// TIA Portal V15.1 export
// export: Created 2020-06-12T07:35:52.2724609Z, ExportSetting None, DisplayName Totally Integrated Automation Portal, DisplayVersion V15.1, DisplayName TIA Portal Openness, DisplayVersion V15.1, DisplayName STEP 7 Professional, DisplayVersion V15.1, DisplayName STEP 7 Safety, DisplayVersion V15.1, DisplayName WinCC Advanced, DisplayVersion V15.1
FUNCTION "MELT_Curves" : Void   // FC224, FBD
TITLE = Melt curves management
{ S7_Optimized_Access := 'FALSE' }
// stored: SetENOAutomatically False
   VAR_TEMP
      tMode : Int;
      tPmax : Real;
      tImax : Real;
      tIdx : Int;
      tDoCheck : Bool;
      tHTRelPower : Real;
      i : Int;
      tX : Real;
      tZ : Real;
      tR : Real;
      tPF : Real;
      tRslag : Real;
      tIset : Real;
      tUmin : Real;
      tUmax : Real;
   END_VAR
BEGIN

REGION Network 1: Staring resistance curve
   // Swing controller will be activatied during start phase, after time delay. After 
   // this the Resistance curve will be frosen
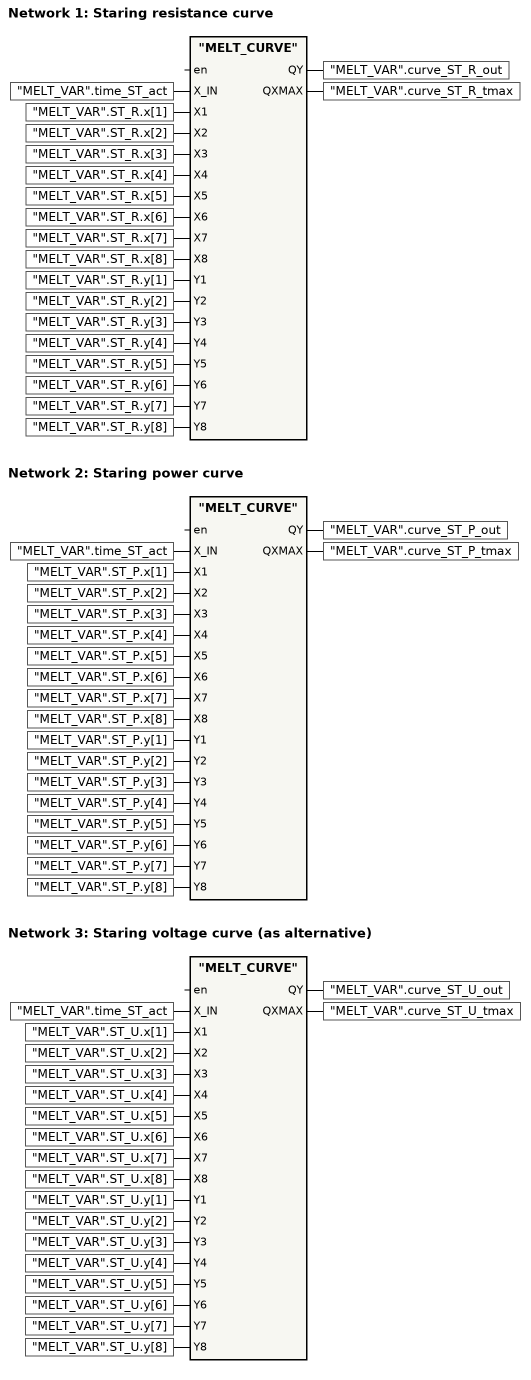
   "MELT_CURVE"(X_IN := "MELT_VAR".time_ST_act,
                X1 := "MELT_VAR".ST_R.x[1],
                X2 := "MELT_VAR".ST_R.x[2],
                X3 := "MELT_VAR".ST_R.x[3],
                X4 := "MELT_VAR".ST_R.x[4],
                X5 := "MELT_VAR".ST_R.x[5],
                X6 := "MELT_VAR".ST_R.x[6],
                X7 := "MELT_VAR".ST_R.x[7],
                X8 := "MELT_VAR".ST_R.x[8],
                Y1 := "MELT_VAR".ST_R.y[1],
                Y2 := "MELT_VAR".ST_R.y[2],
                Y3 := "MELT_VAR".ST_R.y[3],
                Y4 := "MELT_VAR".ST_R.y[4],
                Y5 := "MELT_VAR".ST_R.y[5],
                Y6 := "MELT_VAR".ST_R.y[6],
                Y7 := "MELT_VAR".ST_R.y[7],
                Y8 := "MELT_VAR".ST_R.y[8],
                QY => "MELT_VAR".curve_ST_R_out,
                QXMAX => "MELT_VAR".curve_ST_R_tmax);
END_REGION

REGION Network 2: Staring power curve
   "MELT_CURVE"(X_IN := "MELT_VAR".time_ST_act,
                X1 := "MELT_VAR".ST_P.x[1],
                X2 := "MELT_VAR".ST_P.x[2],
                X3 := "MELT_VAR".ST_P.x[3],
                X4 := "MELT_VAR".ST_P.x[4],
                X5 := "MELT_VAR".ST_P.x[5],
                X6 := "MELT_VAR".ST_P.x[6],
                X7 := "MELT_VAR".ST_P.x[7],
                X8 := "MELT_VAR".ST_P.x[8],
                Y1 := "MELT_VAR".ST_P.y[1],
                Y2 := "MELT_VAR".ST_P.y[2],
                Y3 := "MELT_VAR".ST_P.y[3],
                Y4 := "MELT_VAR".ST_P.y[4],
                Y5 := "MELT_VAR".ST_P.y[5],
                Y6 := "MELT_VAR".ST_P.y[6],
                Y7 := "MELT_VAR".ST_P.y[7],
                Y8 := "MELT_VAR".ST_P.y[8],
                QY => "MELT_VAR".curve_ST_P_out,
                QXMAX => "MELT_VAR".curve_ST_P_tmax);
END_REGION

REGION Network 3: Staring voltage curve (as alternative)
   "MELT_CURVE"(X_IN := "MELT_VAR".time_ST_act,
                X1 := "MELT_VAR".ST_U.x[1],
                X2 := "MELT_VAR".ST_U.x[2],
                X3 := "MELT_VAR".ST_U.x[3],
                X4 := "MELT_VAR".ST_U.x[4],
                X5 := "MELT_VAR".ST_U.x[5],
                X6 := "MELT_VAR".ST_U.x[6],
                X7 := "MELT_VAR".ST_U.x[7],
                X8 := "MELT_VAR".ST_U.x[8],
                Y1 := "MELT_VAR".ST_U.y[1],
                Y2 := "MELT_VAR".ST_U.y[2],
                Y3 := "MELT_VAR".ST_U.y[3],
                Y4 := "MELT_VAR".ST_U.y[4],
                Y5 := "MELT_VAR".ST_U.y[5],
                Y6 := "MELT_VAR".ST_U.y[6],
                Y7 := "MELT_VAR".ST_U.y[7],
                Y8 := "MELT_VAR".ST_U.y[8],
                QY => "MELT_VAR".curve_ST_U_out,
                QXMAX => "MELT_VAR".curve_ST_U_tmax);
END_REGION

REGION Network 4: Internal inducatnce
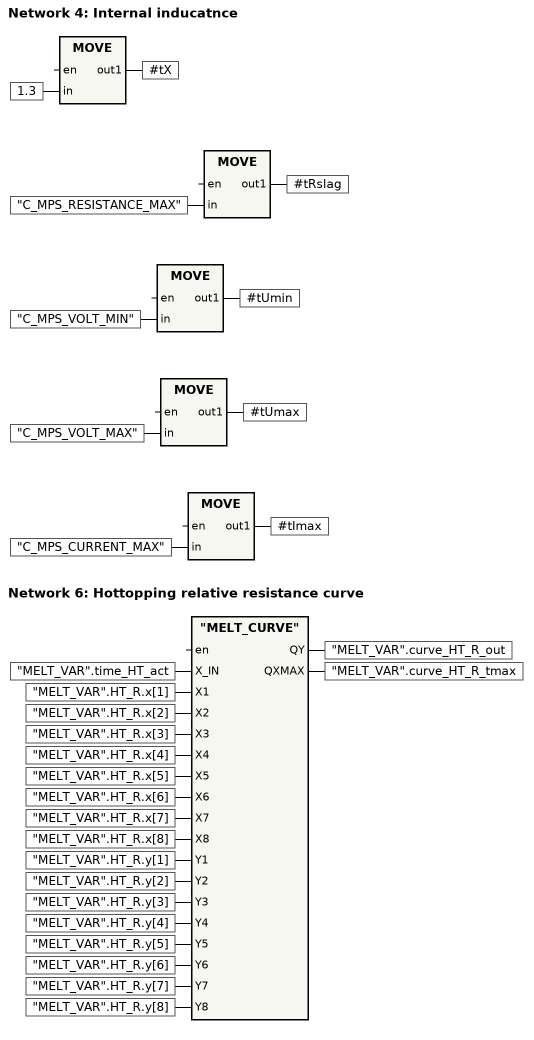
   #tX := 1.3;
   #tRslag := "C_MPS_RESISTANCE_MAX";
   #tUmin := "C_MPS_VOLT_MIN";
   #tUmax := "C_MPS_VOLT_MAX";
   #tImax := "C_MPS_CURRENT_MAX";
END_REGION

REGION Network 5 (SCL): Recaclulate the starting curve: (P,R) -> (U,R)
   IF "MELT_VAR".use_recalc_u THEN
       #tIset := 10.0;
       FOR #i := 1 TO 8 DO
       #tR := "MELT_VAR".ST_R.y[#i];
       #tZ := #tR + #tX;
       #tPF := #tR / #tZ;
       "PUR_CONSTR"(iEnable:=true,
                    iMode:=2,
                    iCosPhi:=#tPF,
                    iRslag:=#tRslag,
                    pQmax:=3500.0,
                    pUmin:=#tUmin,
                    pUmax:=#tUmax,
                    pImax:=#tImax,
                    qPmax=>#tPmax,
                    qImax=>#tImax,
                    ioPset:="MELT_VAR".ST_P.y[#i],
                    ioRset:="MELT_VAR".ST_R.y[#i],
                    ioUset:="MELT_VAR".ST_U.y[#i],
                    ioIset:=#tIset);

       END_FOR;
   END_IF;
END_REGION

REGION Network 6: Hottopping relative resistance curve
   "MELT_CURVE"(X_IN := "MELT_VAR".time_HT_act,
                X1 := "MELT_VAR".HT_R.x[1],
                X2 := "MELT_VAR".HT_R.x[2],
                X3 := "MELT_VAR".HT_R.x[3],
                X4 := "MELT_VAR".HT_R.x[4],
                X5 := "MELT_VAR".HT_R.x[5],
                X6 := "MELT_VAR".HT_R.x[6],
                X7 := "MELT_VAR".HT_R.x[7],
                X8 := "MELT_VAR".HT_R.x[8],
                Y1 := "MELT_VAR".HT_R.y[1],
                Y2 := "MELT_VAR".HT_R.y[2],
                Y3 := "MELT_VAR".HT_R.y[3],
                Y4 := "MELT_VAR".HT_R.y[4],
                Y5 := "MELT_VAR".HT_R.y[5],
                Y6 := "MELT_VAR".HT_R.y[6],
                Y7 := "MELT_VAR".HT_R.y[7],
                Y8 := "MELT_VAR".HT_R.y[8],
                QY => "MELT_VAR".curve_HT_R_out,
                QXMAX => "MELT_VAR".curve_HT_R_tmax);
END_REGION

REGION Network 7: Hottopping relative power curve
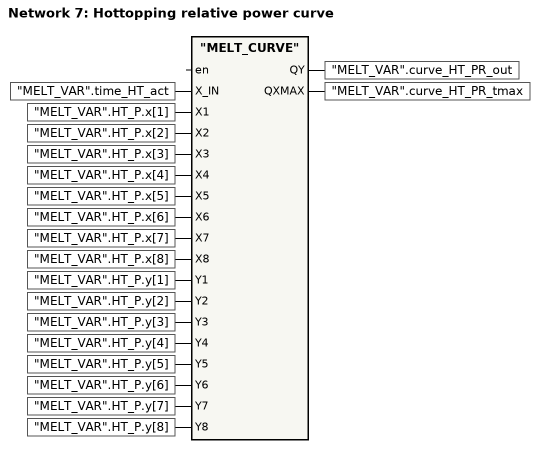
   "MELT_CURVE"(X_IN := "MELT_VAR".time_HT_act,
                X1 := "MELT_VAR".HT_P.x[1],
                X2 := "MELT_VAR".HT_P.x[2],
                X3 := "MELT_VAR".HT_P.x[3],
                X4 := "MELT_VAR".HT_P.x[4],
                X5 := "MELT_VAR".HT_P.x[5],
                X6 := "MELT_VAR".HT_P.x[6],
                X7 := "MELT_VAR".HT_P.x[7],
                X8 := "MELT_VAR".HT_P.x[8],
                Y1 := "MELT_VAR".HT_P.y[1],
                Y2 := "MELT_VAR".HT_P.y[2],
                Y3 := "MELT_VAR".HT_P.y[3],
                Y4 := "MELT_VAR".HT_P.y[4],
                Y5 := "MELT_VAR".HT_P.y[5],
                Y6 := "MELT_VAR".HT_P.y[6],
                Y7 := "MELT_VAR".HT_P.y[7],
                Y8 := "MELT_VAR".HT_P.y[8],
                QY => "MELT_VAR".curve_HT_PR_out,
                QXMAX => "MELT_VAR".curve_HT_PR_tmax);
END_REGION
END_FUNCTION
